{attribute 'qualified_only'}
{attribute 'strict'}
TYPE E_Status :
(
	Off,
	Fault,
	Ready,
	Starting,
	Running,
	Stopping,
	Checking
);
END_TYPE

(* stored: Version 1.1.0.1, ProductVersion 3.1.4026.11
   DUT E_Status: Id {ff422239-7a9a-4fab-aac4-c6bdfa6c8873} *)
